FUNCTION_BLOCK FB_TimeCrossCheck2System
VAR_INPUT
	TimeStruct_Sys1 : TIMESTRUCT;
 	TimeStruct_Sys2 : TIMESTRUCT;
	secondDifferentAllow : UDINT; 
END_VAR
VAR_OUTPUT
	bErrorTimeTwoSystem : BOOL;
END_VAR
VAR
	DtSys1 : DT;
	DtSys2 : DT;
	uDSys1 : LREAL;
	uDsys2 : LREAL;
	diferent : lreal;
	
END_VAR


DtSys1 := SYSTEMTIME_TO_DT(TimeStruct_Sys1);
DtSys2 := SYSTEMTIME_TO_DT(TimeStruct_Sys2);

uDSys1 := DT_TO_LREAL(DtSys1);
uDSys2 := DT_TO_LREAL(DtSys2);
diferent := uDSys1 - uDsys2;
IF ABS(uDSys1 - uDsys2) > secondDifferentAllow THEN
	bErrorTimeTwoSystem := TRUE;
ELSE
	bErrorTimeTwoSystem := FALSE;
END_IF

END_FUNCTION_BLOCK

(* stored: Version 1.1.0.1, ProductVersion 3.1.4024.12
   POU FB_TimeCrossCheck2System: Id {307e072b-510f-4c75-9757-777bcad11ff3}, SpecialFunc None *)
